{attribute 'qualified_only'}
VAR_GLOBAL
	
	doHome : BOOL;
	
END_VAR

(* stored: Version 1.1.0.1, ProductVersion 3.1.4022.17
   GVL COM: Id {34a59a86-ea11-4ac6-84d9-4bbe8ae687ea} *)
